TYPE "Prod_Coil_Ctrl"
VERSION : 0.1
// Block: Prod_Coil_Ctrl
   STRUCT
      Setup_LinePreparation_Exe : Bool;
      STOP_Provino : Bool;
      ACK_Provino : Bool;
      STOP_Taglio_Fine_Ordini : Bool;
      STOP_Manca_Dati_AspoInLinea : Bool;
      STOP_Manca_Dati_AspoInCarico : Bool;
      STOP_FineTurno : Bool;
      STOP_ControlloQualita : Bool;
   END_STRUCT;

END_TYPE
